TYPE ST_JOB_INFO :
STRUCT
	sPartNumber:	T_MaxString;
	sRevision:		T_MaxString;
	sJobNumber:		T_MaxString;
END_STRUCT
END_TYPE

(* stored: Version 1.1.0.1, ProductVersion 3.1.4024.12
   DUT ST_JOB_INFO: Id {1e6b70b2-d5b3-4c70-82ef-762c1a922099} *)
